// TIA Portal V17 export
// export: Created 2024-08-20T10:59:44.833072Z, ExportSetting WithDefaults, DisplayName Totally Integrated Automation Portal, DisplayVersion V17 Update 4, DisplayName TIA Portal Openness, DisplayVersion V17 Update 4, DisplayName TIA Portal Version Control Interface, DisplayVersion V17, DisplayName STEP 7 Professional, DisplayVersion V17 Update 4, DisplayName STEP 7 Safety, DisplayVersion V17, DisplayName WinCC Advanced, DisplayVersion V17 Update 4
VAR_GLOBAL   // PLC tag table "IO"
   PCM_EEE_EMER AT %I0.0 : Bool;   // PCM-E-CF-01-04 BOTAO DE EMERGENCIA - ATUADO
   PCM_EEE_K27 AT %I0.1 : Bool;   // PCM-E-CF-01-04 RELE DE PROTECAO FUNCAO 27 - ATUADO
   PCM_EEE_DJL AT %I0.2 : Bool;   // PCM-E-CF-01-04 DISJUNTOR GERAL STATUS - LIGADO
   PCM_EEE_DJD AT %I0.3 : Bool;   // PCM-E-CF-01-04 DISJUNTOR GERAL STATUS - DESLIGADO
   PCM_EEE_DJYFAL AT %I0.4 : Bool;   // PCM-E-CF-01-04 DISJUNTOR GERAL STATUS - FALHA
   PCM_EEE_DJFG AT %I0.5 : Bool;   // PCM-E-CF-01-04 FALHA GERAL ATUADO
   PCM_EEE_TR01_KA3 AT %I0.6 : Bool;   // PCM-E-CF-01-04 TRANSFORMADOR -TR-01 ALARME TEMP 150°
   PCM_EEE_TR01_KA4 AT %I0.7 : Bool;   // PCM-E-CF-01-04 TRANSFORMADOR -TR-01 ALARME TEMP 155°
   PCM_EEE_TR01_KA5 AT %I1.0 : Bool;   // PCM-E-CF-01-04 TRANSFORMADOR -TR-01 FALHA PROTECAO
   PCM_EEE_INTRU AT %I1.1 : Bool;   // PCM-E-CF-01-04 INTRUSAO NO PAINEL (COLUNA 01~04)
   MB_01_FF AT %I1.2 : Bool;   // MB-01 FALTA DE FASE
   MB_01_MMNT AT %I1.3 : Bool;   // MB-01 MODO MANUTENCAO
   MB_01_ML AT %I1.4 : Bool;   // MB-01 MODO LOCAL
   MB_01_MA AT %I1.5 : Bool;   // MB-01 MODO AUTOMATICO
   MB_01_MN AT %I1.6 : Bool;   // MB-01 MODO NORMAL
   MB_01_HMNT AT %I1.7 : Bool;   // MB-01 HABILITA MANUTENCAO
   MB_01_BL AT %I2.0 : Bool;   // MB-01 BOMBA LIGADA
   MB_01_DINV AT %I2.1 : Bool;   // MB-01 DEFEITO NO INVERSOR
   MB_01_DMB AT %I2.2 : Bool;   // MB-01 DEFEITO NA BOMBA
   MB_01_RST AT %I2.3 : Bool;   // MB-01 RESET
   MB_01_INTRU AT %I2.4 : Bool;   // MB-01 INTRUSAO NO PAINEL
   MB_01_EMER AT %I2.5 : Bool;   // MB-01 EMERGENCIA
   MB_02_FF AT %I2.6 : Bool;   // MB-02 FALTA DE FASE
   MB_02_MMNT AT %I2.7 : Bool;   // MB-02 MODO MANUTENCAO
   MB_02_ML AT %I3.0 : Bool;   // MB-02 MODO LOCAL
   MB_02_MA AT %I3.1 : Bool;   // MB-02 MODO AUTOMATICO
   MB_02_MN AT %I3.2 : Bool;   // MB-02 MODO NORMAL
   MB_02_HMNT AT %I3.3 : Bool;   // MB-02 HABILITA MANUTENCAO
   MB_02_BL AT %I3.4 : Bool;   // MB-02 BOMBA LIGADA
   MB_02_DINV AT %I3.5 : Bool;   // MB-02 DEFEITO NO INVERSOR
   MB_02_DMB AT %I3.6 : Bool;   // MB-02 DEFEITO NA BOMBA
   MB_02_RST AT %I3.7 : Bool;   // MB-02 RESET
   MB_02_INTRU AT %I4.0 : Bool;   // MB-02 INTRUSAO NO PAINEL
   MB_02_EMER AT %I4.1 : Bool;   // MB-02 EMERGENCIA
   MB_03_FF AT %I4.2 : Bool;   // MB-03 FALTA DE FASE
   MB_03_MMNT AT %I4.3 : Bool;   // MB-03 MODO MANUTENCAO
   MB_03_ML AT %I4.4 : Bool;   // MB-03 MODO LOCAL
   MB_03_MA AT %I4.5 : Bool;   // MB-03 MODO AUTOMATICO
   MB_03_MN AT %I4.6 : Bool;   // MB-03 MODO NORMAL
   MB_03_HMNT AT %I4.7 : Bool;   // MB-03 HABILITA MANUTENCAO
   MB_03_BL AT %I5.0 : Bool;   // MB-03 BOMBA LIGADA
   MB_03_DINV AT %I5.1 : Bool;   // MB-03 DEFEITO NO INVERSOR
   MB_03_DMB AT %I5.2 : Bool;   // MB-03 DEFEITO NA BOMBA
   MB_03_RST AT %I5.3 : Bool;   // MB-03 RESET
   MB_03_INTRU AT %I5.4 : Bool;   // MB-03 INTRUSAO NO PAINEL
   MB_03_EMER AT %I5.5 : Bool;   // MB-03EMERGENCIA
   MB_04_FF AT %I5.6 : Bool;   // MB-04 FALTA DE FASE
   MB_04_MMNT AT %I5.7 : Bool;   // MB-04 MODO MANUTENCAO
   MB_04_ML AT %I6.0 : Bool;   // MB-04 MODO LOCAL
   MB_04_MA AT %I6.1 : Bool;   // MB-04 MODO AUTOMATICO
   MB_04_MN AT %I6.2 : Bool;   // MB-04 MODO NORMAL
   MB_04_HMNT AT %I6.3 : Bool;   // MB-04 HABILITA MANUTENCAO
   MB_04_BL AT %I6.4 : Bool;   // MB-04 BOMBA LIGADA
   MB_04_DINV AT %I6.5 : Bool;   // MB-04 DEFEITO NO INVERSOR
   MB_04_DMB AT %I6.6 : Bool;   // MB-04 DEFEITO NA BOMBA
   MB_04_RST AT %I6.7 : Bool;   // MB-04 RESET
   MB_04_INTRU AT %I7.0 : Bool;   // MB-04 INTRUSAO NO PAINEL
   MB_04_EMER AT %I7.1 : Bool;   // MB-04 EMERGENCIA
   QGBT_EMER AT %I7.2 : Bool;   // QGBT-AUX-01 BOTAO DE EMERGENCIA ATUADO
   QGBT_K27 AT %I7.3 : Bool;   // QGBT-AUX-01 RELE DE PROTECAO FUNCAO 27/59 ATUADO
   QGBT_DISJ_LIG AT %I7.4 : Bool;   // QGBT-AUX-01 DISJUNTOR GERAL STATUS - LIGADO
   QGBT_DISJ_DESLIG AT %I7.5 : Bool;   // QGBT-AUX-01 DISJUNTOR GERAL STATUS - DESLIGADO
   QGBT_DISJ_YFAL AT %I7.6 : Bool;   // QGBT-AUX-01 DISJUNTOR GERAL FALHA - TRIP
   QGBT_INTRU AT %I7.7 : Bool;   // QGBT-AUX-01 INTRUSAO NO PAINEL
   KI165 AT %I8.0 : Bool;   // RESERVA
   KI166 AT %I8.1 : Bool;   // RESERVA
   KI167 AT %I8.2 : Bool;   // RESERVA
   KI168 AT %I8.3 : Bool;   // RESERVA
   KI169 AT %I8.4 : Bool;   // RESERVA
   KI170 AT %I8.5 : Bool;   // RESERVA
   KI171 AT %I8.6 : Bool;   // RESERVA
   KI172 AT %I8.7 : Bool;   // RESERVA
   LSL_001 AT %I9.0 : Bool;   // CHAVE DE NIVEL -LSL-001
   LSH_001 AT %I9.1 : Bool;   // CHAVE DE NIVEL -LSH-001
   LSL_002 AT %I9.2 : Bool;   // CHAVE DE NIVEL -LSL-002
   LSH_002 AT %I9.3 : Bool;   // CHAVE DE NIVEL -LSH-002
   PCE_EEE_INTRU AT %I9.4 : Bool;   // INTRUSAO NO PAINEL
   PCE_EEE_UPS_ALM AT %I9.5 : Bool;   // UPS EM ALARME FALHA NA BATERIA
   PCE_EEE_UPS_FE AT %I9.6 : Bool;   // UPS EM OPERACAO FALTA DE ENERGIA
   PCE_EEE_UPS_CHAR AT %I9.7 : Bool;   // UPS EM ALARME BATERIA CARREGADA
   MB_01_SH AT %Q0.0 : Bool;   // MB-01 SOLICITACAO HIDRAULICA
   MB_01_PH AT %Q0.1 : Bool;   // MB-01 PROTECAO HIDRAULICA
   MB_01_INTV AT %Q0.2 : Bool;   // MB-01 INTERVALO (COM)
   MB_01_RR AT %Q0.3 : Bool;   // MB-01 RESET REMOTO
   MB_01_INTVS AT %Q0.4 : Bool;   // MB-01 INTERVALO SINAL
   MB_02_SH AT %Q0.5 : Bool;   // MB-02 SOLICITACAO HIDRAULICA
   MB_02_PH AT %Q0.6 : Bool;   // MB-02 PROTECAO HIDRAULICA
   MB_02_INTV AT %Q0.7 : Bool;   // MB-02 INTERVALO (COM)
   MB_02_RR AT %Q1.0 : Bool;   // MB-02 RESET REMOTO
   MB_02_INTVS AT %Q1.1 : Bool;   // MB-02 INTERVALO SINAL
   MB_03_SH AT %Q1.2 : Bool;   // MB-03 SOLICITACAO HIDRAULICA
   MB_03_PH AT %Q1.3 : Bool;   // MB-03 PROTECAO HIDRAULICA
   MB_03_INTV AT %Q1.4 : Bool;   // MB-03 INTERVALO (COM)
   MB_03_RR AT %Q1.5 : Bool;   // MB-03 RESET REMOTO
   MB_03_INTVS AT %Q1.6 : Bool;   // MB-03 INTERVALO SINAL
   MB_04_SH AT %Q1.7 : Bool;   // MB-04 SOLICITACAO HIDRAULICA
   LIT_001 AT %IW10 : Int;   // -LIT-001 TRANSMISSOR DE NIVEL TANQUE (TIPO RADAR)
   MB_01_REF_VEL AT %IW12 : Int;   // REFERENCIA DE VELOCIDADE INVERSOR DE FREQUENCIA BOMBA 01
   MB_02_REF_VEL AT %IW14 : Int;   // REFERENCIA DE VELOCIDADE INVERSOR DE FREQUENCIA BOMBA 02
   MB_03_REF_VEL AT %IW16 : Int;   // REFERENCIA DE VELOCIDADE INVERSOR DE FREQUENCIA BOMBA 03
   MB_04_REF_VEL AT %IW18 : Int;   // REFERENCIA DE VELOCIDADE INVERSOR DE FREQUENCIA BOMBA 04
   FB6 AT %IW20 : Int;   // RESERVA
   FB7 AT %IW22 : Int;   // RESERVA
   FB8 AT %IW24 : Int;   // RESERVA
   FB9 AT %IW26 : Int;   // RESERVA
   FB10 AT %IW28 : Int;   // RESERVA
   FB11 AT %IW30 : Int;   // RESERVA
   FB12 AT %IW32 : Int;   // RESERVA
   FB13 AT %IW34 : Int;   // RESERVA
   FB14 AT %IW36 : Int;   // RESERVA
   FB15 AT %IW38 : Int;   // RESERVA
   FB16 AT %IW40 : Int;   // RESERVA
   MB_01_VEL AT %QW4 : Int;   // SETPOINT INVERSOR DE FREQUENCIA BOMBA 01
   MB_02_VEL AT %QW6 : Int;   // SETPOINT INVERSOR DE FREQUENCIA BOMBA 02
   MB_03_VEL AT %QW8 : Int;   // SETPOINT INVERSOR DE FREQUENCIA BOMBA 03
   MB_04_VEL AT %QW10 : Int;   // SETPOINT INVERSOR DE FREQUENCIA BOMBA 04
   F25 AT %QW12 : Int;   // RESERVA
   F26 AT %QW14 : Int;   // RESERVA
   F27 AT %QW16 : Int;   // RESERVA
   F28 AT %QW18 : Int;   // RESERVA
   MB_04_PH AT %Q2.0 : Bool;   // MB-04 PROTECAO HIDRAULICA
   MB_04_INTV AT %Q2.1 : Bool;   // MB-04 INTERVALO (COM)
   MB_04_RR AT %Q2.2 : Bool;   // MB-04 RESET REMOTO
   MB_04_INTVS AT %Q2.3 : Bool;   // MB-04 INTERVALO SINAL
   KO21 AT %Q2.4 : Bool;   // RESERVA
   KO22 AT %Q2.5 : Bool;   // RESERVA
   KO23 AT %Q2.6 : Bool;   // RESERVA
   KO24 AT %Q2.7 : Bool;   // RESERVA
   KO25 AT %Q3.0 : Bool;   // RESERVA
   KO26 AT %Q3.1 : Bool;   // RESERVA
   KO27 AT %Q3.2 : Bool;   // RESERVA
   KO28 AT %Q3.3 : Bool;   // RESERVA
   KO29 AT %Q3.4 : Bool;   // RESERVA
   KO30 AT %Q3.5 : Bool;   // RESERVA
   KO31 AT %Q3.6 : Bool;   // RESERVA
   KO32 AT %Q3.7 : Bool;   // RESERVA
END_VAR
